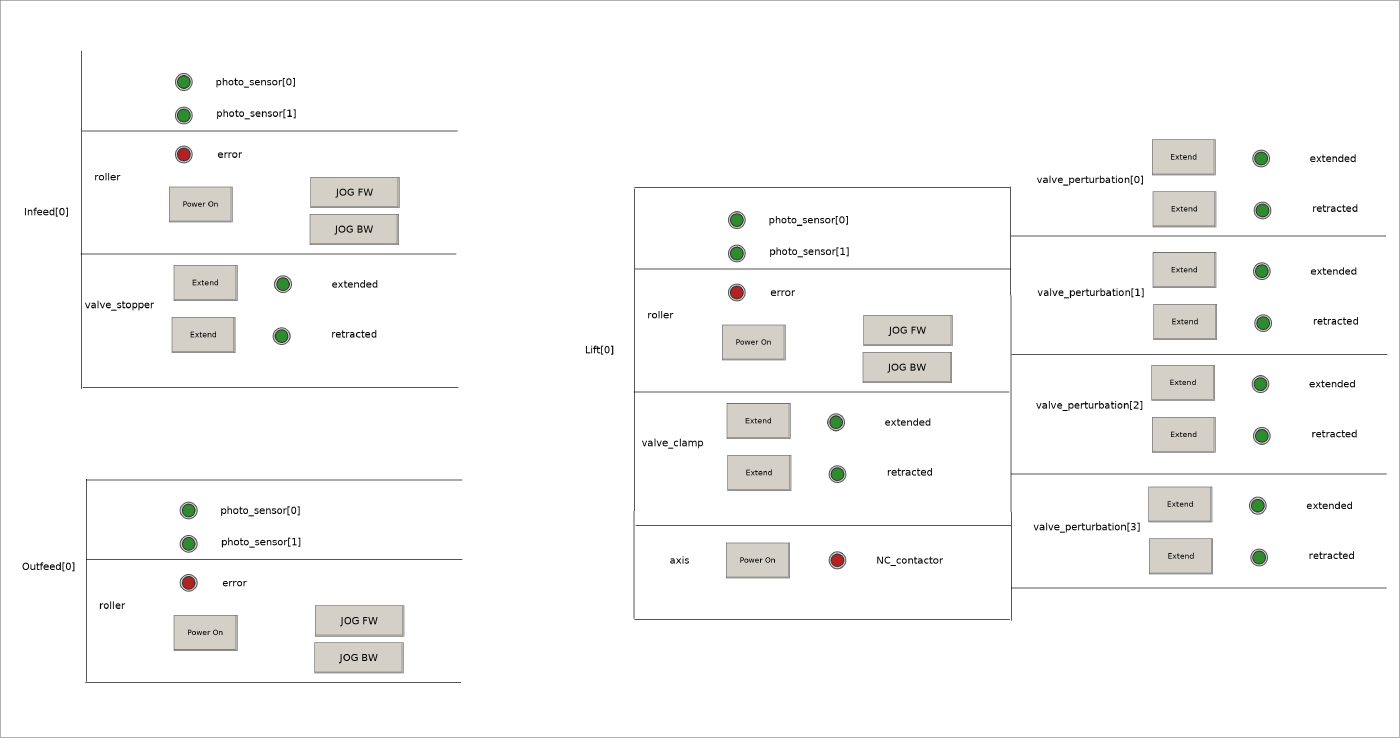
VISUALIZATION v_rem_0  // 2048x1080
VAR_IN_OUT
	dIO_ReM		: Replenishment_Module;
END_VAR
    Lamp1 (254,105 30x30), variable: dIO_ReM.infeed[0].photo_sensor[0].debounced_input.Q, style: Lamp-Lamp1-Green
    Lamp1 (254,154 30x30), variable: dIO_ReM.infeed[0].photo_sensor[1].debounced_input.Q, style: Lamp-Lamp1-Green
    Label (308,107 132x26), "photo_sensor[0]"
    Label (309,153 132x26), "photo_sensor[1]"
    Label (28,297 80x26), "Infeed[0]"
    Lamp1 (254,211 30x30), variable: dIO_ReM.infeed[0].roller.err, style: Lamp-Lamp1-Red
    Label (270,213 132x26), "error"
    Label (91,246 132x26), "roller"
    Line (120,191) (669,191)
    Line (119,74) (119,569)
    Label (109,433 132x26), "valve_stopper"
    Button (454,259 130x45), "JOG FW", colour toggle: dIO_ReM.infeed[0].roller.forward
        OnMouseDown: execute { dIO_ReM.infeed[0].roller.forward := TRUE; }
        OnMouseUp: execute { dIO_ReM.infeed[0].roller.forward := FALSE; }
    Button (453,313 130x45), "JOG BW", colour toggle: dIO_ReM.infeed[0].roller.backward
        OnMouseDown: execute { dIO_ReM.infeed[0].roller.backward := TRUE; }
        OnMouseUp: execute { dIO_ReM.infeed[0].roller.backward := FALSE; }
    Button (247,273 93x52), "Power On", colour toggle: dIO_ReM.infeed[0].roller.Power
        toggle dIO_ReM.infeed[0].roller.Power
    Button (254,388 93x52), "Extend", colour toggle: dIO_ReM.infeed[0].valve_stopper.extend
        OnMouseDown: execute { dIO_ReM.infeed[0].valve_stopper.extend := TRUE; dIO_ReM.infeed[0].valve_stopper.retract := FALSE; }
    Button (251,464 93x52), "Extend", colour toggle: dIO_ReM.infeed[0].valve_stopper.retract
        OnMouseDown: execute { dIO_ReM.infeed[0].valve_stopper.extend := FALSE; dIO_ReM.infeed[0].valve_stopper.retract := TRUE; }
    Lamp1 (399,401 30x30), variable: dIO_ReM.infeed[0].valve_stopper.extended, style: Lamp-Lamp1-Green
    Lamp1 (397,477 30x30), variable: dIO_ReM.infeed[0].valve_stopper.retracted, style: Lamp-Lamp1-Green
    Label (453,403 132x26), "extended"
    Label (452,476 132x26), "retracted"
    Line (118,371) (667,371)
    Line (121,567) (670,567)
    Lamp1 (261,732 30x30), variable: dIO_ReM.outfeed[0].photo_sensor[0].debounced_input.Q, style: Lamp-Lamp1-Green
    Lamp1 (261,781 30x30), variable: dIO_ReM.outfeed[0].photo_sensor[1].debounced_input.Q, style: Lamp-Lamp1-Green
    Label (315,734 132x26), "photo_sensor[0]"
    Label (316,780 132x26), "photo_sensor[1]"
    Label (31,816 80x26), "Outfeed[0]"
    Lamp1 (261,838 30x30), variable: dIO_ReM.outfeed[0].roller.err, style: Lamp-Lamp1-Red
    Label (277,840 132x26), "error"
    Label (98,873 132x26), "roller"
    Line (127,818) (676,818)
    Line (126,701) (126,997)
    Button (461,886 130x45), "JOG FW", colour toggle: dIO_ReM.outfeed[0].roller.forward
        OnMouseDown: execute { dIO_ReM.outfeed[0].roller.forward := TRUE; }
        OnMouseUp: execute { dIO_ReM.outfeed[0].roller.forward := FALSE; }
    Button (460,940 130x45), "JOG BW", colour toggle: dIO_ReM.outfeed[0].roller.backward
        OnMouseDown: execute { dIO_ReM.outfeed[0].roller.backward := TRUE; }
        OnMouseUp: execute { dIO_ReM.outfeed[0].roller.backward := FALSE; }
    Button (254,900 93x52), "Power On", colour toggle: dIO_ReM.outfeed[0].roller.Power
        toggle dIO_ReM.outfeed[0].roller.Power
    Line (125,998) (674,998)
    Line (127,702) (676,702)
    Lamp1 (1063,307 30x30), variable: dIO_ReM.lift[0].photo_sensor[0].debounced_input.Q, style: Lamp-Lamp1-Green
    Lamp1 (1063,356 30x30), variable: dIO_ReM.lift[0].photo_sensor[1].debounced_input.Q, style: Lamp-Lamp1-Green
    Label (1117,309 132x26), "photo_sensor[0]"
    Label (1118,355 132x26), "photo_sensor[1]"
    Label (837,499 80x26), "Lift[0]"
    Lamp1 (1063,413 30x30), variable: dIO_ReM.lift[0].roller.err, style: Lamp-Lamp1-Red
    Label (1079,415 132x26), "error"
    Label (900,448 132x26), "roller"
    Line (929,393) (1478,393)
    Line (928,276) (927,905)
    Label (918,635 132x26), "valve_clamp"
    Button (1263,461 130x45), "JOG FW", colour toggle: dIO_ReM.lift[0].roller.forward
        OnMouseDown: execute { dIO_ReM.lift[0].roller.forward := TRUE; }
        OnMouseUp: execute { dIO_ReM.lift[0].roller.forward := FALSE; }
    Button (1262,515 130x45), "JOG BW", colour toggle: dIO_ReM.lift[0].roller.backward
        OnMouseDown: execute { dIO_ReM.lift[0].roller.backward := TRUE; }
        OnMouseUp: execute { dIO_ReM.lift[0].roller.backward := FALSE; }
    Button (1056,475 93x52), "Power On", colour toggle: dIO_ReM.lift[0].roller.Power
        toggle dIO_ReM.lift[0].roller.Power
    Button (1063,590 93x52), "Extend", colour toggle: dIO_ReM.lift[0].valve_clamp.extend
        OnMouseDown: execute { dIO_ReM.lift[0].valve_clamp.extend := TRUE; dIO_ReM.lift[0].valve_clamp.retract := FALSE; }
    Button (1064,666 93x52), "Extend", colour toggle: dIO_ReM.lift[0].valve_clamp.retract
        OnMouseDown: execute { dIO_ReM.lift[0].valve_clamp.extend := FALSE; dIO_ReM.lift[0].valve_clamp.retract := TRUE; }
    Lamp1 (1208,603 30x30), variable: dIO_ReM.lift[0].valve_clamp.extended, style: Lamp-Lamp1-Green
    Lamp1 (1210,679 30x30), variable: dIO_ReM.lift[0].valve_clamp.retracted, style: Lamp-Lamp1-Green
    Label (1262,605 132x26), "extended"
    Label (1265,678 132x26), "retracted"
    Line (927,573) (1476,573)
    Line (930,769) (1479,769)
    Label (1515,250 160x26), "valve_perturbation[0]"
    Button (1685,204 93x52), "Extend", colour toggle: dIO_ReM.lift[0].valve_perturbation[0].extend
        OnMouseDown: execute { dIO_ReM.lift[0].valve_perturbation[0].extend := TRUE; dIO_ReM.lift[0].valve_perturbation[0].retract := FALSE; }
    Button (1686,280 93x52), "Extend", colour toggle: dIO_ReM.lift[0].valve_perturbation[0].retract
        OnMouseDown: execute { dIO_ReM.lift[0].valve_perturbation[0].extend := FALSE; dIO_ReM.lift[0].valve_perturbation[0].retract := TRUE; }
    Lamp1 (1830,217 30x30), variable: dIO_ReM.lift[0].valve_perturbation[0].extended, style: Lamp-Lamp1-Green
    Lamp1 (1832,293 30x30), variable: dIO_ReM.lift[0].valve_perturbation[0].retracted, style: Lamp-Lamp1-Green
    Label (1884,219 132x26), "extended"
    Label (1887,292 132x26), "retracted"
    Label (1516,415 160x26), "valve_perturbation[1]"
    Button (1686,369 93x52), "Extend", colour toggle: dIO_ReM.lift[0].valve_perturbation[1].extend
        OnMouseDown: execute { dIO_ReM.lift[0].valve_perturbation[1].extend := TRUE; dIO_ReM.lift[0].valve_perturbation[1].retract := FALSE; }
    Button (1687,445 93x52), "Extend", colour toggle: dIO_ReM.lift[0].valve_perturbation[1].retract
        OnMouseDown: execute { dIO_ReM.lift[0].valve_perturbation[1].extend := FALSE; dIO_ReM.lift[0].valve_perturbation[1].retract := TRUE; }
    Lamp1 (1831,382 30x30), variable: dIO_ReM.lift[0].valve_perturbation[1].extended, style: Lamp-Lamp1-Green
    Lamp1 (1833,458 30x30), variable: dIO_ReM.lift[0].valve_perturbation[1].retracted, style: Lamp-Lamp1-Green
    Label (1885,384 132x26), "extended"
    Label (1888,457 132x26), "retracted"
    Label (1514,580 160x26), "valve_perturbation[2]"
    Button (1684,534 93x52), "Extend", colour toggle: dIO_ReM.lift[0].valve_perturbation[2].extend
        OnMouseDown: execute { dIO_ReM.lift[0].valve_perturbation[2].extend := TRUE; dIO_ReM.lift[0].valve_perturbation[2].retract := FALSE; }
    Button (1685,610 93x52), "Extend", colour toggle: dIO_ReM.lift[0].valve_perturbation[2].retract
        OnMouseDown: execute { dIO_ReM.lift[0].valve_perturbation[2].extend := FALSE; dIO_ReM.lift[0].valve_perturbation[2].retract := TRUE; }
    Lamp1 (1829,547 30x30), variable: dIO_ReM.lift[0].valve_perturbation[2].extended, style: Lamp-Lamp1-Green
    Lamp1 (1831,623 30x30), variable: dIO_ReM.lift[0].valve_perturbation[2].retracted, style: Lamp-Lamp1-Green
    Label (1883,549 132x26), "extended"
    Label (1886,622 132x26), "retracted"
    Label (1510,758 160x26), "valve_perturbation[3]"
    Button (1680,712 93x52), "Extend", colour toggle: dIO_ReM.lift[0].valve_perturbation[3].extend
        OnMouseDown: execute { dIO_ReM.lift[0].valve_perturbation[3].extend := TRUE; dIO_ReM.lift[0].valve_perturbation[3].retract := FALSE; }
    Button (1681,788 93x52), "Extend", colour toggle: dIO_ReM.lift[0].valve_perturbation[3].retract
        OnMouseDown: execute { dIO_ReM.lift[0].valve_perturbation[3].extend := FALSE; dIO_ReM.lift[0].valve_perturbation[3].retract := TRUE; }
    Lamp1 (1825,725 30x30), variable: dIO_ReM.lift[0].valve_perturbation[3].extended, style: Lamp-Lamp1-Green
    Lamp1 (1827,801 30x30), variable: dIO_ReM.lift[0].valve_perturbation[3].retracted, style: Lamp-Lamp1-Green
    Label (1879,727 132x26), "extended"
    Label (1882,800 132x26), "retracted"
    Line (1478,273) (1479,908)
    Line (1478,345) (2027,345)
    Line (1480,518) (2029,518)
    Line (1479,693) (2028,693)
    Line (1479,860) (2028,860)
    Line (928,274) (1477,274)
    Line (928,906) (1477,906)
    Label (1265,807 132x26), "NC_contactor"
    Label (928,807 132x26), "axis"
    Button (1062,794 93x52), "Power On", colour toggle: dIO_ReM.lift[0].power_axis
        toggle dIO_ReM.lift[0].power_axis
    Lamp1 (1210,805 30x30), variable: dIO_ReM.lift[0].contactor_axis, style: Lamp-Lamp1-Red
END_VISUALIZATION

(* stored: Version 1.1.0.1, ProductVersion 3.1.4024.12
   Visu v_rem_0: Id {5c93d195-e8bd-46c5-b6cb-5d024bd76eab} *)
